// TIA Portal V16 export
// export: Created 2021-06-11T21:02:52.7612225Z, ExportSetting WithDefaults, DisplayName Totally Integrated Automation Portal, DisplayVersion V16 Update 4, DisplayName TIA Portal Version Control Interface, DisplayVersion V16 Update 2, DisplayName TIA Portal Openness, DisplayVersion V16 Update 4, DisplayName SINAMICS Startdrive Advanced, DisplayVersion V16 Update 5, DisplayName SINAMICS Startdrive G130, G150, S120, S150, SINAMICS MV, S210, DisplayVersion V16 Update 5, DisplayName SINAMICS Startdrive G110M, G120, G120C, G120D, G120P, G115D, DisplayVersion V16 Update 5, DisplayName STEP 7 Professional, DisplayVersion V16 Update 4, DisplayName STEP 7 Safety, DisplayVersion V16, DisplayName WinCC Advanced / Unified PC, DisplayVersion V16 Update 4, DisplayName WinCC Unified LineCoordination, DisplayVersion V16, DisplayName WinCC Unified Sequence, DisplayVersion V16
FUNCTION_BLOCK "fb_ContactorControl"   // FB1, LAD
{ S7_Optimized_Access := 'TRUE' }
VERSION : 0.1
// stored: AutoNumber true, IsIECCheckEnabled false, IsRetainMemResEnabled false, MemoryReserve 100, SetENOAutomatically false, UDAEnableTagReadback false
   VAR_INPUT
      interlock : Bool;
      overload : Bool;
      stopPB : Bool;
      resetPB : Bool;
   END_VAR
   VAR_OUTPUT
      contactor : Bool;
      status : Int;
      resetCMD : Bool;
   END_VAR
   VAR_IN_OUT
      startPB : Bool;
      jogPB : Bool;
   END_VAR
BEGIN

REGION Network 1
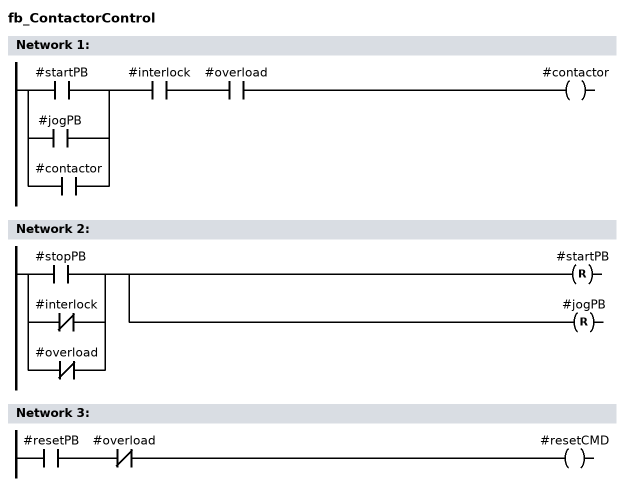
   RUNG wire#powerrail
      Contact( #startPB )
      wire#w1
      Contact( #interlock )
      Contact( #overload )
      Coil( #contactor )
   END_RUNG
   RUNG wire#powerrail
      Contact( #jogPB )
   END_RUNG wire#w1
   RUNG wire#powerrail
      Contact( #contactor )
   END_RUNG wire#w1
   // the same network as SCL:
   #contactor := (#startPB OR #jogPB OR #contactor) AND #interlock AND #overload;
END_REGION

REGION Network 2
   RUNG wire#powerrail
      Contact( #stopPB )
      wire#w1
      R_Coil( #startPB )
   END_RUNG
   RUNG wire#powerrail
      I_Contact( #interlock )
   END_RUNG wire#w1
   RUNG wire#powerrail
      I_Contact( #overload )
   END_RUNG wire#w1
   RUNG wire#w1
      R_Coil( #jogPB )
   END_RUNG
   // the same network as SCL:
   IF #stopPB OR NOT #interlock OR NOT #overload THEN
       #startPB := FALSE;
       #jogPB := FALSE;
   END_IF;
END_REGION

REGION Network 3
   RUNG wire#powerrail
      Contact( #resetPB )
      I_Contact( #overload )
      Coil( #resetCMD )
   END_RUNG
   // the same network as SCL:
   #resetCMD := #resetPB AND NOT #overload;
END_REGION

REGION Network 4 (SCL)
   IF NOT #startPB AND NOT #contactor AND NOT #jogPB AND #overload THEN
       #status := 0;
   ELSIF #startPB AND #contactor AND NOT #jogPB AND #overload THEN
       #status := 1;
   ELSIF NOT #startPB AND #contactor AND #jogPB AND #overload THEN
       #status := 2;
   ELSIF NOT #startPB AND NOT #contactor AND NOT #jogPB AND NOT #overload THEN
       #status := 3;
   END_IF;
END_REGION
END_FUNCTION_BLOCK
